FUNCTION_BLOCK FB_PrintModule_WEU_View
VAR
  // helper
  bInit   : BOOL;
  
  // config
  _pModule : POINTER TO FB_PrintModule_WEU;
  _pPositioning : POINTER TO FB_PrintPositionDmax;
  
  // view selections
  nSelWorkerPrint : UDINT := 1;
  bShowDropSpeedSetup : BOOL;
  // hardware view
  bShowPhDetail : BOOL;
  nSelPhDetail : UDINT := 1;
  bShowPcDetail : BOOL;
  nSelPcDetail : UDINT := 1;
  
  // motion and position
  bShowPositionDetail : BOOL;
  bMovingInd : BOOL;
  fSpeed  : LREAL;
  fbBlink_Moving : FB_BLINK;
  
  fbBlink_Printing : FB_BLINK;
  bBlinkPrint : BOOL;
  bPrintInd : ARRAY[1..GVL_WEU.nC_WorkerPrintPerPm] OF BOOL;
  t : TIME;
  zPos_PM : UDINT;
  i : UDINT;
END_VAR

VAR CONSTANT
  nC_MAX_WORKER_VIEWS : UINT := 10;
END_VAR

IF NOT checkConfig() THEN RETURN; END_IF    // check config

// -- show moving -----------------------
fSpeed := _pPositioning^.getSpeed();
IF LrealIsNaN(x:=fSpeed) THEN
  fSpeed := 0;
END_IF
t := LREAL_TO_TIME(1000-fSpeed*900);
fbBlink_Moving(bI_Enable:=SEL(fSpeed > 0, FALSE, TRUE), tI_Time:=t, bO_Out=>bMovingInd);

t := T#400MS;
fbBlink_Moving(bI_Enable:=TRUE, tI_Time:=t, bO_Out=>bBlinkPrint);
FOR i:=1 TO GVL_WEU.nC_WorkerPrintPerPm DO
  bPrintInd[i] := _pModule^.fbWorkerPrint[i].bPrinting AND bBlinkPrint;
END_FOR


// -- show pm module position
zPos_PM := SEL(_pModule^._pModuleMachineState^.bUnitInPrintPosition, 0, 40);

// -- show ph detail
nSelPhDetail := LIMIT(1, nSelPhDetail, _pModule^._nPh);
nSelPcDetail := LIMIT(1, nSelPcDetail, _pModule^._nPc);

METHOD checkConfig : BOOL
VAR_INPUT
END_VAR
VAR_INST
  _fX_m, _fY_m   : LREAL;
  _nX_px, _nY_px : DINT; 
END_VAR
VAR
  bOK : BOOL;
END_VAR
IF NOT bInit THEN RETURN; END_IF

checkConfig := TRUE;
END_METHOD

METHOD init : BOOL
VAR_INPUT
  pModule : POINTER TO FB_PrintModule_WEU;
  pPositioning : POINTER TO FB_PrintPositionDmax;
END_VAR
IF pPositioning = 0 OR pModule = 0 THEN RETURN; END_IF

_pModule := pModule;
_pPositioning := pPositioning;

bInit := TRUE;
END_METHOD

END_FUNCTION_BLOCK

(* stored: Version 1.1.0.1, ProductVersion 3.1.4024.11
   POU FB_PrintModule_WEU_View: Id {57a6df33-c5fc-4b78-b796-858abcecd4f4}, SpecialFunc None
   Method checkConfig: Id {edfe75ad-63c4-4ec1-9d31-8e206962e7b0}
   Method init: Id {bd002f50-5fd9-48d9-b817-a794ac96eb55} *)
